FUNCTION_BLOCK ADD_INT (* IEC 61131-3 INT Addition *)
  (* Standard: 61131-3 *)
  (* Version 0.0, 2004-12-15, JHC, Rockwell Automation, Converted from SRC format. *)
  (* Compiler header: package fb.rt.plc.math; *)
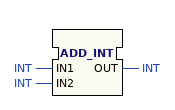
  VAR_INPUT
    IN1 : INT; (* Augend *)
    IN2 : INT; (* Addend *)
  END_VAR
  VAR_OUTPUT
    OUT : INT; (* Sum *)
  END_VAR
END_FUNCTION_BLOCK
